// TIA Portal V16 export
// export: Created 2022-03-04T10:52:05.6814005Z, ExportSetting WithDefaults, DisplayName Totally Integrated Automation Portal, DisplayVersion V16 Update 3, DisplayName TIA Portal Version Control Interface, DisplayVersion V16 Update 2, DisplayName TIA Portal Openness, DisplayVersion V16 Update 3, DisplayName STEP 7 Professional, DisplayVersion V16 Update 3, DisplayName STEP 7 Safety, DisplayVersion V16, DisplayName WinCC Professional, DisplayVersion V16 Update 3
ORGANIZATION_BLOCK "OB00030_IntNCyclic_100ms"   // OB30, LAD, CyclicInterrupt
{ S7_Optimized_Access := 'TRUE' }
VERSION : 0.1
// stored: AutoNumber true, IsIECCheckEnabled false, SetENOAutomatically false
   VAR_INPUT
      Initial_Call : Bool;   // Initial call of this OB
      Event_Count : Int;   // Events discarded
   END_VAR
BEGIN

REGION Network 1: 2nd Order Response Simulation
   // ▀▀▀▀▀▀▀▀▀▀▀▀▀▀▀▀▀▀▀▀▀▀▀▀▀▀▀▀▀▀▀▀▀▀▀▀▀▀▀▀▀▀▀▀
   // Generates (in this case) a unit step response to a second order transfer function
   // ▄▄▄▄▄▄▄▄▄▄▄▄▄▄▄▄▄▄▄▄▄▄▄▄▄▄▄▄▄▄▄▄▄▄▄▄▄▄▄▄▄▄▄▄
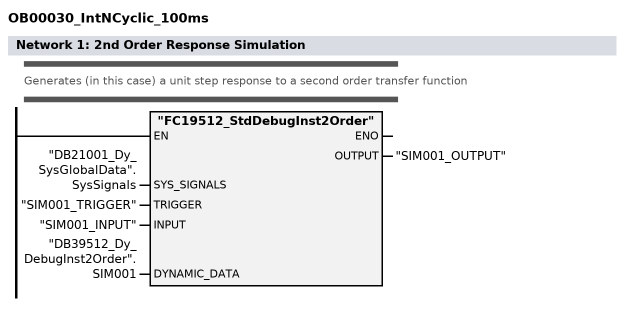
   RUNG wire#powerrail
      "FC19512_StdDebugInst2Order"(SYS_SIGNALS := "DB21001_Dy_SysGlobalData".SysSignals, TRIGGER := "SIM001_TRIGGER", INPUT := "SIM001_INPUT", DYNAMIC_DATA := "DB39512_Dy_DebugInst2Order".SIM001, OUTPUT => "SIM001_OUTPUT")
   END_RUNG
   // the same network as SCL:
   "FC19512_StdDebugInst2Order"(SYS_SIGNALS := "DB21001_Dy_SysGlobalData".SysSignals,
                           TRIGGER := "SIM001_TRIGGER",
                           INPUT := "SIM001_INPUT",
                           DYNAMIC_DATA := "DB39512_Dy_DebugInst2Order".SIM001,
                           OUTPUT => "SIM001_OUTPUT");
END_REGION
END_ORGANIZATION_BLOCK
